Staubli VAL3: Main.pgx

public program Main(num x_nType)
  local num l_nKey
begin
  //
  bUserRefresh=bListRefresh=true
  bExit=false
  nType=x_nType
  //
  do
    call Refresh()
    call RefreshList()
    call user:setList("坐标系",sList,bUserRefresh,bListRefresh,nSelected,sItem,l_nKey)
    bUserRefresh=false
    bListRefresh=false
    call MainKey(l_nKey)
    delay(0)
  until bExit

end
